FUNCTION_BLOCK FB_MqttDeviceTriggerDiscovery EXTENDS FB_MqttDeviceDiscoveryBase
VAR_INPUT
END_VAR
VAR_OUTPUT
END_VAR
VAR
	stConfig : ST_MqttDeviceTriggerConfiguration;
END_VAR

PROPERTY PROTECTED Component : STRING(30)
GET
Component := 'device_automation';
END_GET
END_PROPERTY

METHOD  ConfigToJson : STRING(1000)
VAR_INPUT
END_VAR
VAR
	fbJsonWriter : FB_JsonSaxWriter;
END_VAR
fbJsonWriter.ResetDocument();
fbJsonWriter.StartObject();
fbJsonWriter.AddKeyString(key := 'atype', value := 'trigger');
fbJsonWriter.AddKeyString(key := 'pl', value := stConfig.payload);
fbJsonWriter.AddKeyNumber(key := 'qos', value := stConfig.qos);
fbJsonWriter.AddKeyString(key := 't', value := stConfig.topic);
fbJsonWriter.AddKeyString(key := 'type', value := stConfig.event_type);
fbJsonWriter.AddKeyString(key := 'stype', value := stConfig.event_subtype);
THIS^.DevInfoToJson(fbJsonWriter); 
fbJsonWriter.EndObject();
fbJsonWriter.CopyDocument(pDoc := ConfigToJson, nDoc := 1000);
END_METHOD

PROPERTY PUBLIC Configuration : ST_MqttDeviceTriggerConfiguration
GET
Configuration := THIS^.stConfig;
END_GET
SET
THIS^.stConfig := Configuration;
END_SET
END_PROPERTY

END_FUNCTION_BLOCK

(* stored: Version 1.1.0.1, ProductVersion 3.1.4024.5
   POU FB_MqttDeviceTriggerDiscovery: Id {4c86cbbe-4ac9-4788-b201-7c50d96ffe98}, SpecialFunc None
   Property Component: Id {6bea9714-f3b9-4e0f-9c4d-cd024141adf5}
   Get Get: Id {bbf2f96e-25e6-4090-8a75-bb0d96250629}
   Method ConfigToJson: Id {1ee008b6-f689-4ffa-b15f-3da2ef996a7c}
   Property Configuration: Id {10a29d25-fd76-4ca0-83f2-2659c1b4be8d}
   Get Get: Id {df18c658-0017-47c1-a585-bab4d895b09f}
   Set Set: Id {a12039bb-934b-433e-93af-c7ef7b3c4b7c} *)
